// TIA Portal V20 export
FUNCTION_BLOCK "CentralShifter_Move_Pallets"   // FB19, LAD
{ S7_Optimized_Access := 'TRUE' }
// stored: MemoryReserve 100, SetENOAutomatically false
   VAR
      Motor_Driver_Instance { S7_SetPoint := 'True'} : "Side_Driver";
      Speed : Int := 400;
      Auto_Go_Left : Bool;
      Auto_Go_Right : Bool;
      CSM1_Comm_ok : Bool;
      CSM2_Comm_ok : Bool;
      prevCentering : Bool;
      tCenteringTimer : TON_TIME;
   END_VAR
   VAR_TEMP
      "czujnik lewy" : Bool;
      "czujnik prawy" : Bool;
   END_VAR
BEGIN

REGION Network 1
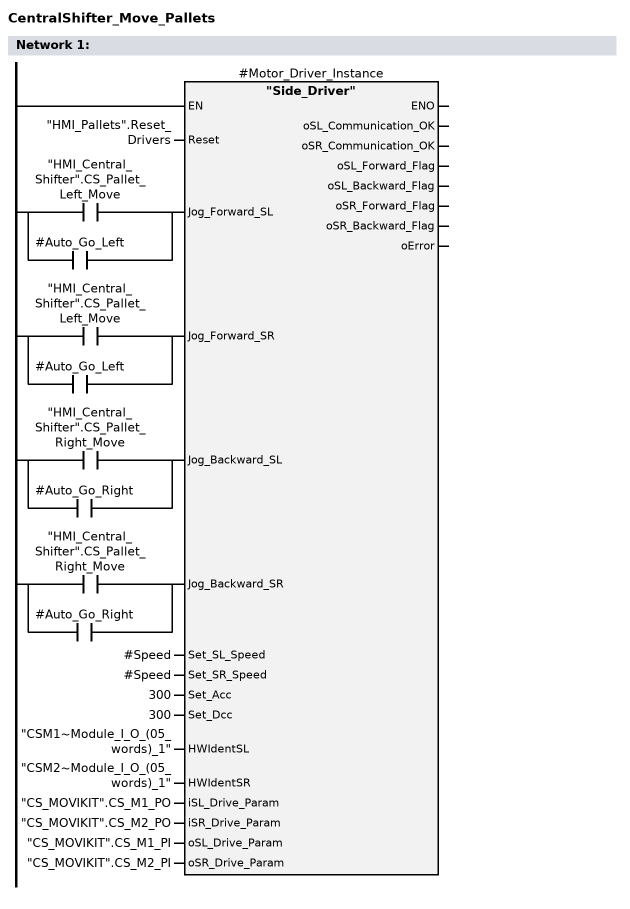
   RUNG wire#powerrail
      #Motor_Driver_Instance(Jog_Forward_SL := wire#w1, Jog_Forward_SR := wire#w2, Jog_Backward_SL := wire#w3, Jog_Backward_SR := wire#w4, Reset := "HMI_Pallets".Reset_Drivers, Set_SL_Speed := #Speed, Set_SR_Speed := #Speed, Set_Acc := 300, Set_Dcc := 300, HWIdentSL := "CSM1~Module_I_O_(05_words)_1", HWIdentSR := "CSM2~Module_I_O_(05_words)_1", iSL_Drive_Param := "CS_MOVIKIT".CS_M1_PO, iSR_Drive_Param := "CS_MOVIKIT".CS_M2_PO, oSL_Drive_Param := "CS_MOVIKIT".CS_M1_PI, oSR_Drive_Param := "CS_MOVIKIT".CS_M2_PI, oSL_Communication_OK =>, oSR_Communication_OK =>, oSL_Forward_Flag =>, oSL_Backward_Flag =>, oSR_Forward_Flag =>, oSR_Backward_Flag =>, oError =>)
   END_RUNG
   RUNG wire#powerrail
      Contact( "HMI_Central_Shifter".CS_Pallet_Left_Move )
   END_RUNG wire#w1
   RUNG wire#powerrail
      Contact( #Auto_Go_Left )
   END_RUNG wire#w1
   RUNG wire#powerrail
      Contact( "HMI_Central_Shifter".CS_Pallet_Left_Move )
   END_RUNG wire#w2
   RUNG wire#powerrail
      Contact( #Auto_Go_Left )
   END_RUNG wire#w2
   RUNG wire#powerrail
      Contact( "HMI_Central_Shifter".CS_Pallet_Right_Move )
   END_RUNG wire#w3
   RUNG wire#powerrail
      Contact( #Auto_Go_Right )
   END_RUNG wire#w3
   RUNG wire#powerrail
      Contact( "HMI_Central_Shifter".CS_Pallet_Right_Move )
   END_RUNG wire#w4
   RUNG wire#powerrail
      Contact( #Auto_Go_Right )
   END_RUNG wire#w4
   // the same network as SCL:
   #Motor_Driver_Instance(Reset := "HMI_Pallets".Reset_Drivers,   // "Side_Driver"
                          Jog_Forward_SL := "HMI_Central_Shifter".CS_Pallet_Left_Move OR #Auto_Go_Left,
                          Jog_Forward_SR := "HMI_Central_Shifter".CS_Pallet_Left_Move OR #Auto_Go_Left,
                          Jog_Backward_SL := "HMI_Central_Shifter".CS_Pallet_Right_Move OR #Auto_Go_Right,
                          Jog_Backward_SR := "HMI_Central_Shifter".CS_Pallet_Right_Move OR #Auto_Go_Right,
                          Set_SL_Speed := #Speed,
                          Set_SR_Speed := #Speed,
                          Set_Acc := 300,
                          Set_Dcc := 300,
                          HWIdentSL := "CSM1~Module_I_O_(05_words)_1",
                          HWIdentSR := "CSM2~Module_I_O_(05_words)_1",
                          iSL_Drive_Param := "CS_MOVIKIT".CS_M1_PO,
                          iSR_Drive_Param := "CS_MOVIKIT".CS_M2_PO,
                          oSL_Drive_Param := "CS_MOVIKIT".CS_M1_PI,
                          oSR_Drive_Param := "CS_MOVIKIT".CS_M2_PI);
END_REGION

REGION Network 2 (SCL)

   // Logika timera — włącza się tylko gdy trwa centrowanie
   #tCenteringTimer(
                   IN := "HMI_Central_Shifter".CS_Pallet_Centering,
                   PT := T#5S
   );


   IF #tCenteringTimer.Q THEN
       "HMI_Central_Shifter".CS_Pallet_Centering := FALSE;
   END_IF;

   // --- Dotychczasowa logika sterowania ---
   IF "HMI_Central_Shifter".CS_Pallet_Centering AND "iCS_SensorHoming_Left" AND NOT "iCS_SensorHoming_Right" THEN
       "HMI_Central_Shifter".CS_Pallet_Left_Move := 0;
       "HMI_Central_Shifter".CS_Pallet_Right_Move := 1;

   ELSIF "HMI_Central_Shifter".CS_Pallet_Centering AND "iCS_SensorHoming_Right" AND NOT "iCS_SensorHoming_Left" THEN
       "HMI_Central_Shifter".CS_Pallet_Left_Move := 1;
       "HMI_Central_Shifter".CS_Pallet_Right_Move := 0;

   ELSIF "HMI_Central_Shifter".CS_Pallet_Centering THEN
       "HMI_Central_Shifter".CS_Pallet_Left_Move := 0;
       "HMI_Central_Shifter".CS_Pallet_Right_Move := 0;
       "HMI_Central_Shifter".CS_Pallet_Centering := 0;
   END_IF;

   IF NOT "HMI_Central_Shifter".CS_Pallet_Centering AND #prevCentering THEN
       // Jednorazowe wyłączenie jazdy w lewo i prawo
       "HMI_Central_Shifter".CS_Pallet_Left_Move := 0;
       "HMI_Central_Shifter".CS_Pallet_Right_Move := 0;
   END_IF;

   // Aktualizacja stanu poprzedniego
   #prevCentering := "HMI_Central_Shifter".CS_Pallet_Centering;
END_REGION
END_FUNCTION_BLOCK
